FUNCTION_BLOCK FB_Betriebsarten
VAR_INPUT
	Start, NotStop, Weiter, Fehler, Start_Init : BOOL;
    Auto_Fertig   : BOOL; // kommt von fbAuto.Automatikbetrieb_Fertig
    Auto_Stoerung : BOOL; // kommt von fbAuto.Stoerung_erkannt
	A2_Requested: BOOL;
	Alt_abort: BOOL;
	Alt_found: BOOL;
	D3_Requested: BOOL;
	Init_reached: BOOL;
	Cycle_ended: BOOL;
	//Reset			: BOOL;
	//Schalter		: BOOL;
	//Schrittkette_GS : BOOL;
END_VAR
VAR_OUTPUT
	A1 : BOOL; //Initialzustand
	A2 : BOOL; //Stillstand angefordert am Ende des Zyklus
//	A3 : BOOL; //Stillstand angefordert in einem bestimmten Zustand
//	A4 : BOOL; //Erhaltener Stillstand
	A5 : BOOL; //Vorbereitung zur Wiederaufnahme nach Störung
	A6 : BOOL; //Fahrt in den Initialzustand
	F1 : BOOL; //Normalbetrieb
//	F2 : BOOL; //Anfahren
//	F3 : BOOL; //Abfahren
	F4 : BOOL; //Handbetrieb
//	F5 : BOOL; //Schrittbetrieb
//	F6 : BOOL; //Testbetrieb
	D1 : BOOL; //Not-Aus
	D2 : BOOL; //DIagnose und Störbehandlung
	D3 : BOOL; //Produktion trotz Störung
END_VAR
VAR
	bFirstScan : BOOL := TRUE;	

	RS_InitialState: RS;	
	RS_InitialDrive: RS;
	RS_ManualOperationMode: RS;
	RS_AutomaticOperationMode: RS;
	RS_CycleEnded: RS;

	R_TRIG_Manual: R_TRIG;
	R_TRIG_Automatic: R_TRIG;
	R_TRIG_InitialDrive: R_TRIG;
	R_TRIG_CycleEnded: R_TRIG;
	R_TRIG_Init: R_TRIG;
	RS_D2: RS;
	RS_F1: RS;
	RS_D1: RS;
	RS_A5: RS;
	RS_A1: RS;

	RS_D3: RS;

	RS_A2: RS;
	RS_A6: RS;
END_VAR

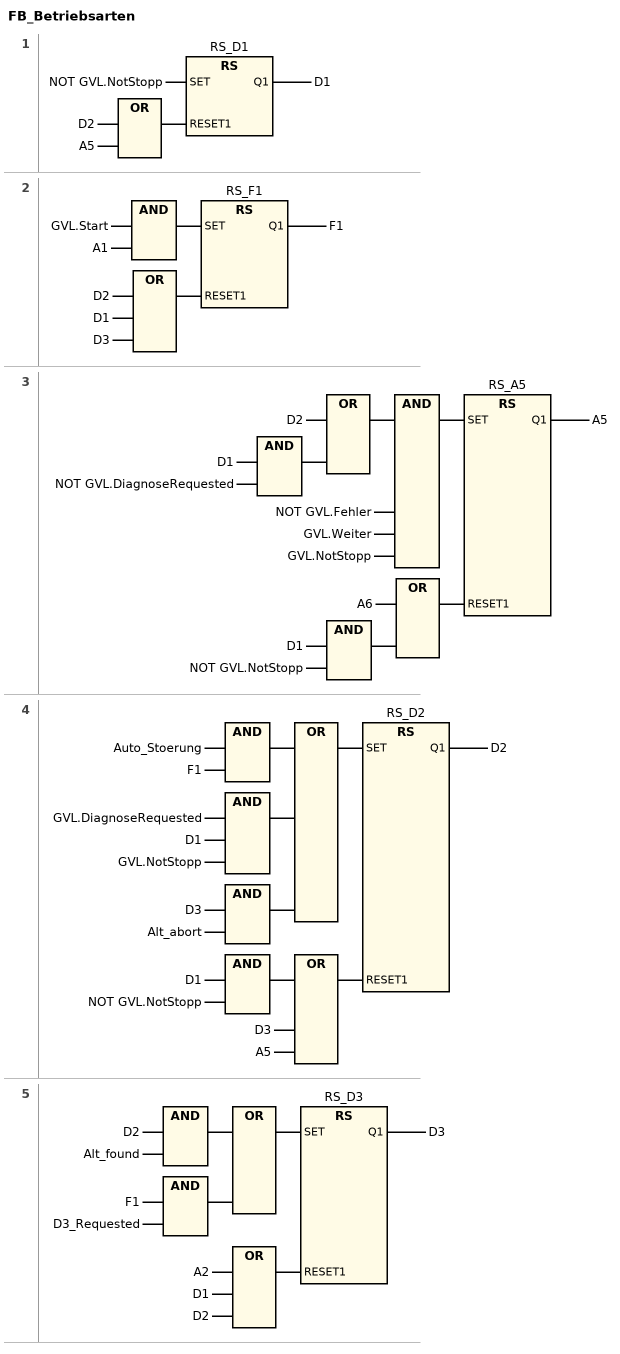
// NETWORK 1
RS_D1(SET := NOT GVL.NotStopp, RESET1 := D2 OR A5); // RS
D1 := RS_D1.Q1;

// NETWORK 2
RS_F1(SET := GVL.Start AND A1, RESET1 := D2 OR D1 OR D3); // RS
F1 := RS_F1.Q1;

// NETWORK 3
RS_A5(SET := (D2 OR D1 AND (NOT GVL.DiagnoseRequested)) AND (NOT GVL.Fehler) AND GVL.Weiter AND GVL.NotStopp, RESET1 := A6 OR D1 AND (NOT GVL.NotStopp)); // RS
A5 := RS_A5.Q1;

// NETWORK 4
RS_D2(SET := Auto_Stoerung AND F1 OR GVL.DiagnoseRequested AND D1 AND GVL.NotStopp OR D3 AND Alt_abort, RESET1 := D1 AND (NOT GVL.NotStopp) OR D3 OR A5); // RS
D2 := RS_D2.Q1;

// NETWORK 5
RS_D3(SET := D2 AND Alt_found OR F1 AND D3_Requested, RESET1 := A2 OR D1 OR D2); // RS
D3 := RS_D3.Q1;

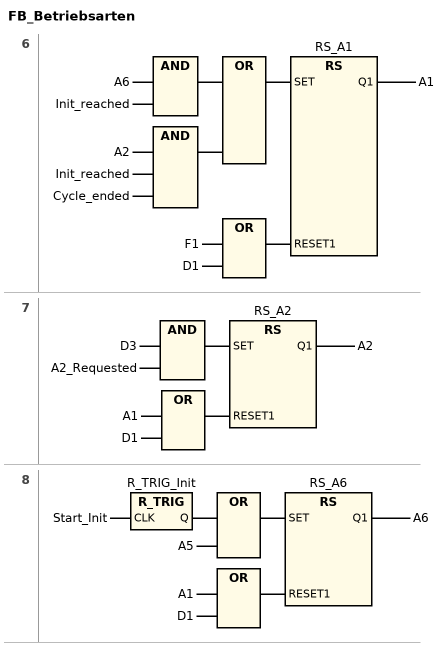
// NETWORK 6
RS_A1(SET := A6 AND Init_reached OR A2 AND Init_reached AND Cycle_ended, RESET1 := F1 OR D1); // RS
A1 := RS_A1.Q1;

// NETWORK 7
RS_A2(SET := D3 AND A2_Requested, RESET1 := A1 OR D1); // RS
A2 := RS_A2.Q1;

// NETWORK 8
R_TRIG_Init(CLK := Start_Init); // R_TRIG
RS_A6(SET := R_TRIG_Init.Q OR A5, RESET1 := A1 OR D1); // RS
A6 := RS_A6.Q1;

END_FUNCTION_BLOCK

(* stored: Version 1.1.0.1
   POU FB_Betriebsarten: Id {06fb9674-c769-4193-84ea-e1b3e704e56b}, SpecialFunc None *)
